FUNCTION_BLOCK fbTask IMPLEMENTS ITask
VAR
	_taskState : eTaskState;
	_component : IComponent;	
END_VAR

PROPERTY Done : BOOL
GET
Done := THIS^._taskState = eTaskState.Done;

IF(Done) THEN
	THIS^._taskState := eTaskState.Idle;
END_IF
END_GET
END_PROPERTY

METHOD DoneWhen 
VAR_INPUT
	Condition : BOOL;
END_VAR
IF (Condition) THEN
	THIS^._taskState := eTaskState.Done;
	_component.Lock := 0;
END_IF;
END_METHOD

METHOD Execute : BOOL
VAR_INPUT
	lockKey : INT;
END_VAR
Execute := (_component.Lock = 0 OR lockKey = _component.Lock) AND_THEN THIS^._taskState = eTaskState.Request;

IF(Execute) THEN
	THIS^._taskState := eTaskState.Executing;
	_component.Lock := lockKey;
ELSE
	THIS^._taskState := eTaskState.Idle;
END_IF;
END_METHOD

METHOD PUBLIC FB_init : BOOL
VAR_INPUT
	bInitRetains : BOOL; // if TRUE, the retain variables are initialized (warm start / cold start)
	bInCopyCode : BOOL;  // if TRUE, the instance afterwards gets moved into the copy code (online change)
	component : IComponent;
END_VAR
_component := component;
END_METHOD

METHOD Invoke
IF(THIS^._taskState < eTaskState.Error) THEN
	THIS^._taskState := eTaskState.Request;
END_IF;
END_METHOD

METHOD Reset
VAR_INPUT
END_VAR
THIS^._taskState := eTaskState.Idle;
END_METHOD

END_FUNCTION_BLOCK

(* stored: Version 1.1.0.1, ProductVersion 3.1.4024.5
   POU fbTask: Id {24034ee3-475d-4338-b4dc-23478f0974a9}, SpecialFunc None
   Property Done: Id {e3ea205b-eb06-42b9-b3d8-63efd5ed6521}
   Get Get: Id {65176686-2db0-4acd-880d-da851e8da10c}
   Method DoneWhen: Id {0e4bb473-b258-4a3f-95b9-bb9741040e56}
   Method Execute: Id {d0212bb0-ffcc-4ef5-806d-394cf6e951a4}
   Method FB_init: Id {a5b60cba-9da0-4e51-9e99-230c8717014e}
   Method Invoke: Id {cc03409d-e0bf-43b3-af7b-1069055f0385}
   Method Reset: Id {afacd00c-5569-431f-be3c-22a90381057d} *)
